PROGRAM MAIN
VAR
	diKapasativSensor1 AT %I* : BOOL ;
	bMinneKapasativSensor1 : BOOL := 0 ;
	diKapasativSensor2 AT %I* : BOOL ;
	bMinneKapasativSensor2 : BOOL := 0 ;
	
	AndMinneKapasitet : BOOL := 0 ;
	OrMinneKapasitet : BOOL := 0;
END_VAR

bMinneKapasativSensor1 := diKapasativSensor1 ;
bMinneKapasativSensor2 := diKapasativSensor2 ;

AndMinneKapasitet := diKapasativSensor1 AND diKapasativSensor2 ;
OrMinneKapasitet := diKapasativSensor1 OR diKapasativSensor2 ;

END_PROGRAM

(* stored: Version 1.1.0.1, ProductVersion 3.1.4024.9
   POU MAIN: Id {71bc25b8-c09e-48ee-9e55-e3aa45d0be0d}, SpecialFunc None *)
